// TwinCAT 3 PLC project ControlBox
// ProgramVersion: 3.1.4023.0
// libraries:
//   Tc2_Standard, * (Beckhoff Automation GmbH)
//   Tc2_System, * (Beckhoff Automation GmbH)
//   Tc3_Module, * (Beckhoff Automation GmbH)
// project tree:
//   Controlbox/Interface/ I_controlbox.TcIO
//   Controlbox/Virtual Controlbox/ FB_realcontrolbox.TcPOU, FB_virtualcontrolbox.TcPOU, FB_Controlbox.TcPOU, FB_JoystickNorm.TcPOU (not stored), FB_VurtualControlBox.TcPOU (not stored), E_Status.TcDUT (not stored), E_Modes.TcDUT, ST_JoystickScaling.TcDUT, task1.TcGVL, Visualization.TcVIS
//   / GlobalTextList.TcGTLO, PlcTask.TcTTO, Visualization Manager.TcVMO (not stored)
//   POUs/ MAIN.TcPOU
// real-time tasks:
//   TASK PlcTask: cycle T#10ms, priority 20, ADS port 350

CONFIGURATION ControlBox
    RESOURCE PLC ON TwinCAT3
        TASK PlcTask(INTERVAL := T#10ms, PRIORITY := 20);
        PROGRAM MAIN WITH PlcTask : MAIN;
    END_RESOURCE
END_CONFIGURATION

// ---- Controlbox/Virtual Controlbox/E_Modes.TcDUT
{attribute 'qualified_only'}
{attribute 'strict'}
TYPE E_Modes :
(
	Off,
	Auto,
	Manual
);
END_TYPE

// ---- Controlbox/Virtual Controlbox/ST_JoystickScaling.TcDUT
TYPE ST_JoystickScaling :
STRUCT
fMaxInputValue:LREAL := 20509.0;
fMinInputValue :LREAL:= 11787.0;
fNeutralInputValue :LREAL:= 16175;
fNeutralDeadband :LREAL:= 50.0;
fMaxOutputValue :LREAL:= 1.0;
fMinOutputValue :LREAL:= -1.0;
fNeutralOutputValue: LREAL := 0.0;
END_STRUCT
END_TYPE

// ---- Controlbox/Virtual Controlbox/task1.TcGVL
{attribute 'qualified_only'}
VAR_GLOBAL
	bStart : BOOL;
	bStop : BOOL;
	bTopSwitch : BOOL;
	bManual : BOOL;
	bOn : BOOL;
	eModeSwitch : E_Modes;
	eModes : E_Modes;
	eState : E_Status;
	eStatus : E_Status;
	fJoystickX : LREAL;
	fJoystickY : LREAL;
	bError : BOOL := FALSE;
	fJoyXNormalized : LREAL;
	fJoyYNormalized : LREAL;
END_VAR

// ---- Controlbox/Interface/I_controlbox.TcIO
INTERFACE I_controlbox

METHOD Buttons
VAR_INPUT
	eModes : E_Modes;
	eState : E_Status;
END_VAR
VAR_OUTPUT
	bStart : BOOL;
	bStop : BOOL;
END_VAR
END_METHOD

METHOD Joystick
VAR_INPUT
	eModes : E_Modes;
	eState : E_Status; 
END_VAR
VAR_OUTPUT
	fJoystickY: LREAL;
	fJoystickX: LREAL; 
END_VAR
END_METHOD

METHOD Lamps
VAR_INPUT
	eModes : E_Modes;
	eState : E_Status;
END_VAR
VAR_OUTPUT
	
END_VAR
END_METHOD

METHOD Mode
VAR_INPUT
END_VAR
VAR_OUTPUT
	eModes : E_Modes; 
END_VAR
END_METHOD

METHOD State
VAR_INPUT
	eModes : E_Modes;
END_VAR
VAR_OUTPUT
	eState : E_Status;	
END_VAR
END_METHOD

END_INTERFACE

// ---- POUs/MAIN.TcPOU
PROGRAM MAIN
VAR
	fbVirtualControlBox : FB_VurtualControlBox;
	fbControlbox : FB_Controlbox;
END_VAR

fbVirtualControlBox();
fbControlbox();

END_PROGRAM

// ---- Controlbox/Virtual Controlbox/FB_Controlbox.TcPOU
FUNCTION_BLOCK FB_Controlbox
VAR_INPUT
END_VAR
VAR_OUTPUT
	eModes : E_Modes;
	eState : E_Status;
END_VAR
VAR
	fbJoystickScaled : FB_JoystickNorm;
	fbVirtualcontrolbox : FB_virtualcontrolbox; 
	fbSelectedControlbox : I_controlbox := fbVirtualcontrolbox;
END_VAR


fbJoystickScaled( fRawInput := task1.fJoystickX, fOutput => task1.fJoyXNormalized);
fbJoystickScaled( fRawInput := task1.fJoystickY, fOutput => task1.fJoyYNormalized);


fbSelectedControlbox.Mode(eModes => eModes);

fbSelectedControlbox.State(eModes := eModes, eState=>task1.eState);

END_FUNCTION_BLOCK

// ---- Controlbox/Virtual Controlbox/FB_virtualcontrolbox.TcPOU
FUNCTION_BLOCK FB_virtualcontrolbox IMPLEMENTS I_controlbox
VAR_INPUT
END_VAR
VAR_OUTPUT
END_VAR
VAR
END_VAR

{warning 'add method implementation '}
METHOD Buttons
VAR_INPUT
	eModes	: E_Modes;
	eState	: E_Status;
END_VAR
VAR_OUTPUT
	bStart	: BOOL;
	bStop	: BOOL;
END_VAR
END_METHOD

{warning 'add method implementation '}
METHOD Joystick
VAR_INPUT
	eModes	: E_Modes;
	eState	: E_Status;
END_VAR
VAR_OUTPUT
	fJoystickY	: LREAL;
	fJoystickX	: LREAL;
END_VAR
IF task1.eModeSwitch = E_Modes.Manual AND task1.eStatus = E_Status.Running THEN
	fJoystickY := task1.fJoystickY;
	fJoystickX := task1.fJoystickX;
	
ELSE
	fJoystickY := 0.0;
	fJoystickX := 0.0;
END_IF
END_METHOD

{warning 'add method implementation '}
METHOD Lamps
VAR_INPUT
	eModes	: E_Modes;
	eState	: E_Status;
END_VAR
END_METHOD

{warning 'add method implementation '}
METHOD Mode
VAR_OUTPUT
	eModes	: E_Modes;
END_VAR
CASE eModes OF    
	E_Modes.Off:
		IF task1.bManual AND task1.bOn THEN
			eModes := E_Modes.Manual;
		ELSIF NOT(task1.bManual) AND task1.bOn THEN
			eModes := E_Modes.Auto;
		END_IF
	E_Modes.Auto:
		IF NOT(task1.bOn) THEN
			eModes := E_Modes.Off;
		ELSIF task1.bManual AND task1.bOn THEN
			eModes := E_Modes.Manual;
		END_IF
	E_Modes.Manual:
		IF NOT(task1.bOn) THEN
			eModes := E_Modes.Off;
		ELSIF NOT(task1.bManual) AND task1.bOn THEN
			eModes := E_Modes.Auto;
		END_IF
ELSE
		eModes := E_Modes.Off;
END_CASE
END_METHOD

{warning 'add method implementation '}
METHOD State
VAR_INPUT
	eModes	: E_Modes;
END_VAR
VAR_OUTPUT
	eState	: E_Status;
END_VAR
CASE eState OF
	E_Status.Fault:									
		IF NOT(task1.bError) THEN
			eState := E_Status.Ready;       
		ELSIF eModes = E_Modes.Off THEN
			eState := E_Status.NotReady;
		END_IF										
	E_Status.NotReady:
		IF eModes = E_Modes.Manual OR eModes = E_modes.Auto THEN 
			eState := E_Status.Ready;
		END_IF
	E_Status.Ready:										
		IF task1.bStart THEN
			eState:= E_Status.Starting;
		ELSIF task1.bError THEN
			eState := E_Status.Fault;
		ELSIF eModes = E_Modes.Off THEN
			eState := E_Status.NotReady;
		END_IF
	E_Status.Running:								
		IF task1.bError THEN
			eState := E_Status.Fault;
		ELSIF eModes = E_Modes.Manual AND NOT(task1.bStop) THEN
			task1.bStart:=TRUE;
		ELSIF eModes = E_Modes.Auto AND NOT(task1.bStart) THEN
			eState:= E_Status.Ready;
		ELSIF eModes = E_Modes.Off THEN
			eState := E_Status.NotReady;
		ELSIF task1.bStop THEN
			task1.bStart:=FALSE;			
			eState := E_Status.Stopping;

		END_IF
	E_Status.Starting:							
		eState:= E_Status.Running;
		IF task1.bError THEN
			eState := E_Status.Fault;
		ELSIF eModes = E_Modes.Off THEN
			eState := E_Status.NotReady;
		END_IF
	E_Status.Stopping:							
		eState := E_Status.Ready;
		IF task1.bError THEN
			eState := E_Status.Fault;
		ELSIF eModes = E_Modes.Off THEN
			eState := E_Status.NotReady;
		END_IF
ELSE
	eState := E_Status.NotReady;
END_CASE
END_METHOD

END_FUNCTION_BLOCK

// ---- Controlbox/Virtual Controlbox/FB_realcontrolbox.TcPOU
FUNCTION_BLOCK FB_realcontrolbox IMPLEMENTS I_controlbox
VAR_INPUT
END_VAR
VAR_OUTPUT
END_VAR
VAR
END_VAR

{warning 'add method implementation '}
METHOD Buttons
VAR_INPUT
	eModes	: E_Modes;
	eState	: E_States;
END_VAR
VAR_OUTPUT
	bStart	: BOOL;
	bStop	: BOOL;
END_VAR
END_METHOD

{warning 'add method implementation '}
METHOD Joystick
VAR_INPUT
	eModes	: E_Modes;
	eState	: E_Status;
END_VAR
VAR_OUTPUT
	fJoystickY	: LREAL;
	fJoystickX	: LREAL;
END_VAR
END_METHOD

{warning 'add method implementation '}
METHOD Lamps
VAR_INPUT
	eModes	: E_Modes;
	eState	: E_States;
END_VAR
END_METHOD

{warning 'add method implementation '}
METHOD Mode
VAR_OUTPUT
	eModes	: E_Modes;
END_VAR
END_METHOD

{warning 'add method implementation '}
METHOD State
VAR_INPUT
	eModes	: E_Modes;
END_VAR
VAR_OUTPUT
	eState	: E_States;
END_VAR
END_METHOD

END_FUNCTION_BLOCK

// ---- GlobalTextList.TcGTLO
TEXTLIST GlobalTextList
  83 = '%e'
  168 = '%s'
  240 = '%task1.eStatus'
  996 = 'AUTO'
  995 = 'Auto'
  13 = 'Fault'
  897 = 'HMI '
  991 = 'Hydraulic winch'
  898 = 'JOY X'
  726 = 'JOY Y'
  620 = 'Joystick X'
  84 = 'Joystick Y'
  682 = 'Joystixk X'
  632 = 'MANUAL'
  136 = 'Manual'
  356 = 'Mode'
  423 = 'Mode:'
  974 = 'ON'
  317 = 'Running'
  880 = 'Start'
  96 = 'Status'
  881 = 'Status:'
  947 = 'Stop'
  291 = 'Topswitch'
  176 = 'Topswitch Winch'
END_TEXTLIST

// ---- Controlbox/Virtual Controlbox/Visualization.TcVIS
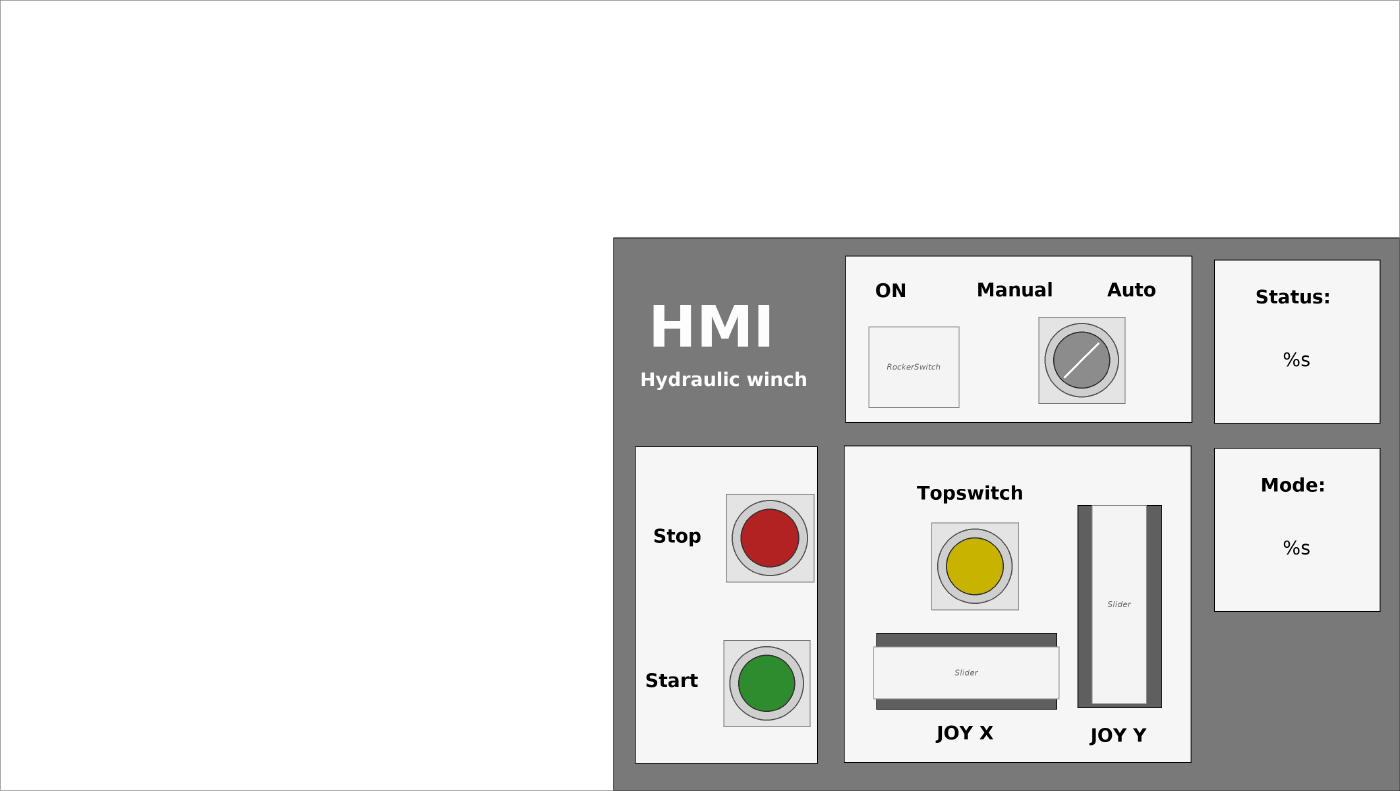
VISUALIZATION Visualization  // 1762x996
    Rectangle (772,299 990x697)
    RoundedRectangle (1528,327 209x206)
    RoundedRectangle (799,562 230x399)
    RoundedRectangle (1062,561 437x399)
    RoundedRectangle (1064,322 436x210)
    PushSwitch (899,622 140x111), variable: task1.bStop, behaviour: TAP, style: Switch-PushSwitch-Red
    PushSwitch (901,806 128x109), variable: task1.bStart, behaviour: TAP, style: Switch-PushSwitch-Green
    Label (774,815 143x84), "Start"
    Label (781,633 143x84), "Stop"
    RockerSwitch (1093,411 114x102), variable: task1.bOn, behaviour: TOGGLE, style: Switch-RockerSwitch-Gray
    RotarySwitch (1295,399 133x109), variable: task1.bManual, behaviour: TOGGLE, style: Switch-RotarySwitch-Gray
    PushSwitch (1171,658 112x110), variable: task1.bTopSwitch, behaviour: TOGGLE, style: Switch-PushSwitch-Yellow
    Label (1146,606 150x30), "Topswitch"
    Label (1333,909 150x34), "JOY Y"
    RoundedRectangle (1356,636 106x255)
    Slider (1374,636 69x250), variable: task1.fJoystickY, scale 11787..20509
    Label (1140,908 150x30), "JOY X"
    RoundedRectangle (1168,732 96x227), angle 270
    Slider (1099,814 234x66), variable: task1.fJoystickX, scale 11787..20509
    Label (1050,324 143x84), "ON"
    Label (1206,323 143x84), "Manual"
    Label (1353,323 143x84), "Auto"
    Label (792,367 232x88), "HMI"
    Label (795,434 232x88), "Hydraulic winch"
    Textfield (1557,438 150x30), "%s", text variable: task1.eStatus
    Label (1556,332 143x84), "Status:"
    RoundedRectangle (1528,564 209x206)
    Textfield (1557,675 150x30), "%s", text variable: task1.eModeSwitch
    Label (1556,569 143x84), "Mode:"
END_VISUALIZATION
